Universal Robots URScript: command05.urscript

def leanForwardLinear():
  movel([0.03490658504,-2.225294796,-1.675516082,-0.7941248097,1.570796327,1.588249619], a=3.0, v=0.8)
  movel([0.3665191429,-2.234021443,-1.658062789,-0.8028514559,1.570796327,1.919862177], a=3.0, v=0.8)
  movel([0.4537856055,-2.00712864,-2.059488517,-0.6457718232,1.570796327,2.024581932], a=3.0, v=0.8)
end
